SUBAPPLICATION PAGE_2 (* Subapplication Type *)
  (* Standard: 61499-2 *)
  (* Version 1.0, 2023-02-07, franz *)
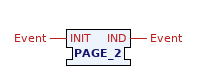
  EVENT_INPUT
    INIT;
  END_EVENT
  EVENT_OUTPUT
    IND;
  END_EVENT
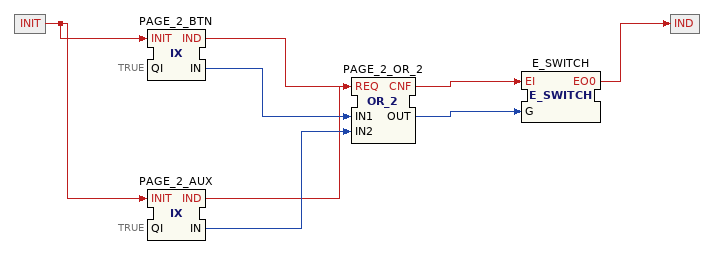
  FBS
    PAGE_2_BTN : IX(QI := TRUE);
    PAGE_2_AUX : IX(QI := TRUE);
    PAGE_2_OR_2 : OR_2;
    E_SWITCH : E_SWITCH;
  END_FBS
  EVENT_CONNECTIONS
    INIT TO PAGE_2_BTN.INIT;
    INIT TO PAGE_2_AUX.INIT;
    PAGE_2_BTN.IND TO PAGE_2_OR_2.REQ;
    PAGE_2_AUX.IND TO PAGE_2_OR_2.REQ;
    PAGE_2_OR_2.CNF TO E_SWITCH.EI;
    E_SWITCH.EO0 TO IND;
  END_CONNECTIONS
  DATA_CONNECTIONS
    PAGE_2_BTN.IN TO PAGE_2_OR_2.IN1;
    PAGE_2_AUX.IN TO PAGE_2_OR_2.IN2;
    PAGE_2_OR_2.OUT TO E_SWITCH.G;
  END_CONNECTIONS
END_SUBAPPLICATION
